KUKA KRL program: wkz1_ok.src, wkz1_ok.dat

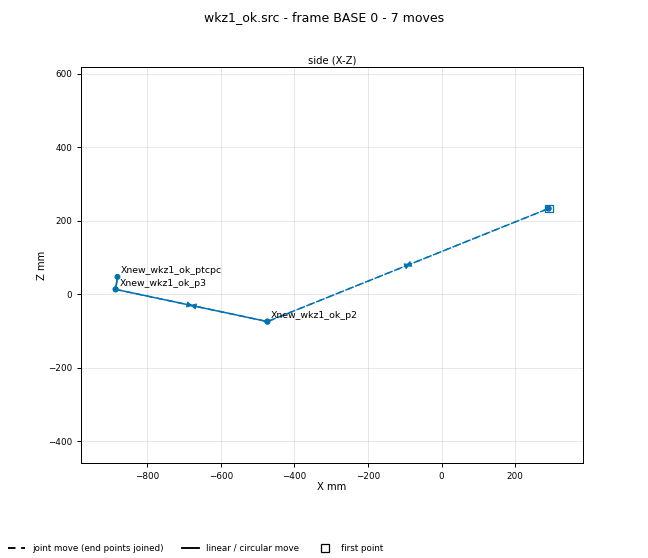
[picture p0: tool path of wkz1_ok.src in frame BASE 0, 7 of 9 moves have a stored position in this frame; points joined in program order, loops and branches not executed]
--- wkz1_ok.src ---
&ACCESS RVP
&COMMENT CHK_TCP_C1
&PARAM DISKPATH = Program/FUNCIONANDO
DEF WKZ1_OK ( )

;# Include block for krc/r1/mada/$config.dat or r1/$config.dat
;# TOOL_DATA[1]={X 73.860,Y 19.790,Z 1095.269,A -165.0000,B -25.0000,C 180.0000}
;# End of Include block for krc/r1/mada/$config.dat or r1/$config.dat
;FOLD INI
  ;FOLD BASISTECH INI
    GLOBAL INTERRUPT DECL 3 WHEN $STOPMESS==TRUE DO IR_STOPM ( )
    INTERRUPT ON 3
    BAS (#INITMOV,0 )
  ;ENDFOLD (BASISTECH INI)
  ;FOLD USER INI
    ;Make your modifications here
  ;ENDFOLD (USER INI)
;ENDFOLD (INI)
;FOLD PTP HOME  Vel= 100 % DEFAULT;%{PE}%V3.2.0,%MKUKATPBASIS,%CMOVE,%VPTP,%P 1:PTP, 2:HOME, 3:, 5:100, 7:DEFAULT
$BWDSTART = FALSE
$H_POS=XHOME
PDAT_ACT=PDEFAULT
BAS (#PTP_DAT )
FDAT_ACT=FHOME
BAS (#FRAMES )
BAS (#VEL_PTP,100 )
PTP  XHOME
;ENDFOLD
;#END_HEADER

;# ============ START PATH : wkz1_ok =============

; Caracterização dos meios de produção:
; Versão Atual:
; 04/05/2013 12:00 Name: P13.090-R6 CHANGES: Check TCP C1
chk_w1_wechs_ok ( )              ; CHECK GUN C1
;FOLD PTP new_wkz1_ok_p1  Vel=100 % P_OLP1 Tool[1]" " Base[0]  ;%{PE}%R8.3,%MKUKATPBASIS,%CMOVE,%VPTP,%P 1:PTP, 2:new_wkz1_ok_p1, 3:, 5:100, 7:P_OLP1
$BWDSTART = FALSE
PDAT_ACT= PP_OLP1
FDAT_ACT= Fnew_wkz1_ok_p1
BAS(#PTP_PARAMS,100)
PTP Xnew_wkz1_ok_p1
;ENDFOLD
;FOLD PTP new_wkz1_ok_p2  Vel=100 % P_OLP2 Tool[1]" " Base[0]  ;%{PE}%R8.3,%MKUKATPBASIS,%CMOVE,%VPTP,%P 1:PTP, 2:new_wkz1_ok_p2, 3:, 5:100, 7:P_OLP2
$BWDSTART = FALSE
PDAT_ACT= PP_OLP2
FDAT_ACT= Fnew_wkz1_ok_p2
BAS(#PTP_PARAMS,100)
PTP Xnew_wkz1_ok_p2
;ENDFOLD
;FOLD LIN new_wkz1_ok_p3  Vel=2.00 m/s L_OLP1 Tool[1]" " Base[0] ;%{PE}%R8.3,%MKUKATPBASIS,%CMOVE,%VLIN,%P 1:LIN, 2:new_wkz1_ok_p3, 3:, 5:2.00, 7:L_OLP1
$BWDSTART = FALSE
LDAT_ACT= LL_OLP1
FDAT_ACT= Fnew_wkz1_ok_p3
BAS(#CP_PARAMS,2.00)
LIN Xnew_wkz1_ok_p3
;ENDFOLD
;Ponto Check TCP
;FOLD LIN new_wkz1_ok_ptcpc  Vel=2.00 m/s L_OLP2 Tool[1]" " Base[0] ;%{PE}%R8.3,%MKUKATPBASIS,%CMOVE,%VLIN,%P 1:LIN, 2:new_wkz1_ok_ptcpc, 3:, 5:2.00, 7:L_OLP2
$BWDSTART = FALSE
LDAT_ACT= LL_OLP2
FDAT_ACT= Fnew_wkz1_ok_ptcpc
BAS(#CP_PARAMS,2.00)
LIN Xnew_wkz1_ok_ptcpc
;ENDFOLD
;FOLD WAIT Time= 3 sec;%{PE}%R8.3,%MKUKATPBASIS,%CWAIT,%VWAIT,%P 2:3
WAIT SEC 3
;ENDFOLD
;FOLD LIN new_wkz1_ok_p4  Vel=2.00 m/s L_OLP3 Tool[1]" " Base[0] ;%{PE}%R8.3,%MKUKATPBASIS,%CMOVE,%VLIN,%P 1:LIN, 2:new_wkz1_ok_p4, 3:, 5:2.00, 7:L_OLP3
$BWDSTART = FALSE
LDAT_ACT= LL_OLP3
FDAT_ACT= Fnew_wkz1_ok_p4
BAS(#CP_PARAMS,2.00)
LIN Xnew_wkz1_ok_p4
;ENDFOLD
;FOLD PTP new_wkz1_ok_p5  Vel=100 % P_OLP3 Tool[1]" " Base[0]  ;%{PE}%R8.3,%MKUKATPBASIS,%CMOVE,%VPTP,%P 1:PTP, 2:new_wkz1_ok_p5, 3:, 5:100, 7:P_OLP3
$BWDSTART = FALSE
PDAT_ACT= PP_OLP3
FDAT_ACT= Fnew_wkz1_ok_p5
BAS(#PTP_PARAMS,100)
PTP Xnew_wkz1_ok_p5
;ENDFOLD
;FOLD PTP new_wkz1_ok_p6  Vel=100 % P_OLP4 Tool[1]" " Base[0]  ;%{PE}%R8.3,%MKUKATPBASIS,%CMOVE,%VPTP,%P 1:PTP, 2:new_wkz1_ok_p6, 3:, 5:100, 7:P_OLP4
$BWDSTART = FALSE
PDAT_ACT= PP_OLP4
FDAT_ACT= Fnew_wkz1_ok_p6
BAS(#PTP_PARAMS,100)
PTP Xnew_wkz1_ok_p6
;ENDFOLD

;#START_TRAILER
;FOLD PTP HOME  Vel= 100 % DEFAULT;%{PE}%V3.2.0,%MKUKATPBASIS,%CMOVE,%VPTP,%P 1:PTP, 2:HOME, 3:, 5:100, 7:DEFAULT
$BWDSTART = FALSE
$H_POS=XHOME
PDAT_ACT=PDEFAULT
BAS (#PTP_DAT )
FDAT_ACT=FHOME
BAS (#FRAMES )
BAS (#VEL_PTP,100 )
PTP  XHOME
;ENDFOLD
END

--- wkz1_ok.dat ---
&ACCESS RVP
&COMMENT CHK_TCP_C1
&PARAM DISKPATH = Program/FUNCIONANDO
DEFDAT  wkz1_ok
;FOLD EXTERNAL DECLARATIONS;%{PE}%MKUKATPBASIS,%CEXT,%VCOMMON,%P
;FOLD BASISTECH EXT;%{PE}%MKUKATPBASIS,%CEXT,%VEXT,%P
EXT  BAS (BAS_COMMAND  :IN,REAL  :IN )
DECL INT SUCCESS
;ENDFOLD (BASISTECH EXT)
;FOLD USER EXT;%{E}%MKUKATPUSER,%CEXT,%VEXT,%P
;Make your modifications here
;ENDFOLD (USER EXT)
;ENDFOLD (EXTERNAL DECLARATIONS)

;# ============ START PATH : wkz1_ok =============
DECL FDAT Fnew_wkz1_ok_p1={TOOL_NO 1,BASE_NO 0,IPO_FRAME #BASE,POINT2[] " "}
DECL PDAT PP_OLP1={VEL 100.0,ACC 50.0,APO_DIST 0.0}
DECL E6POS Xnew_wkz1_ok_p1={X 291.243988,Y -1285.88794,Z 233.281006,A 13.0198002,B 2.4052,C 1.18589997,S 2,T 10}
DECL FDAT Fnew_wkz1_ok_p2={TOOL_NO 1,BASE_NO 0,IPO_FRAME #BASE,POINT2[] " "}
DECL PDAT PP_OLP2={VEL 100.0,ACC 50.0,APO_DIST 0.0}
DECL E6POS Xnew_wkz1_ok_p2={X -473.602997,Y -1280.02002,Z -74.2460022,A 146.021698,B -0.95389998,C -2.53250003,S 2,T 2}
DECL FDAT Fnew_wkz1_ok_p3={TOOL_NO 1,BASE_NO 0,IPO_FRAME #BASE,POINT2[] " "}
DECL E6POS Xnew_wkz1_ok_p3={X -886.51001,Y -1289.66003,Z 13.3669996,A 171.756897,B -2.65339994,C -0.53549999,S 2,T 2}
DECL LDAT LL_OLP1={VEL 2.0,ACC 100.0,APO_DIST 0.0,APO_FAC 0.0,ORI_TYP #VAR,CIRC_TYP #BASE,JERK_FAC 50.0}
DECL FDAT Fnew_wkz1_ok_ptcpc={TOOL_NO 1,BASE_NO 0,IPO_FRAME #BASE,POINT2[] " "}
DECL E6POS Xnew_wkz1_ok_ptcpc={X -881.550415,Y -1291.69397,Z 47.3409119,A 171.412704,B -2.65365791,C -0.829671085,S 18,T 2,E1 0.0,E2 0.0,E3 0.0,E4 0.0,E5 0.0,E6 0.0}
DECL LDAT LL_OLP2={VEL 2.0,ACC 100.0,APO_DIST 0.0,APO_FAC 0.0,ORI_TYP #VAR,CIRC_TYP #BASE,JERK_FAC 50.0}
DECL FDAT Fnew_wkz1_ok_p4={TOOL_NO 1,BASE_NO 0,IPO_FRAME #BASE,POINT2[] " "}
DECL E6POS Xnew_wkz1_ok_p4={X -886.51001,Y -1289.66003,Z 13.3669996,A 171.756897,B -2.65339994,C -0.53549999,S 2,T 2}
DECL LDAT LL_OLP3={VEL 2.0,ACC 100.0,APO_DIST 0.0,APO_FAC 0.0,ORI_TYP #VAR,CIRC_TYP #BASE,JERK_FAC 50.0}
DECL FDAT Fnew_wkz1_ok_p5={TOOL_NO 1,BASE_NO 0,IPO_FRAME #BASE,POINT2[] " "}
DECL PDAT PP_OLP3={VEL 100.0,ACC 50.0,APO_DIST 0.0}
DECL E6POS Xnew_wkz1_ok_p5={X -473.602997,Y -1280.02002,Z -74.2460022,A 146.021698,B -0.95389998,C -2.53250003,S 2,T 2}
DECL FDAT Fnew_wkz1_ok_p6={TOOL_NO 1,BASE_NO 0,IPO_FRAME #BASE,POINT2[] " "}
DECL PDAT PP_OLP4={VEL 100.0,ACC 50.0,APO_DIST 0.0}
DECL E6POS Xnew_wkz1_ok_p6={X 291.243988,Y -1285.88794,Z 233.281006,A 13.0198002,B 2.4052,C 1.18589997,S 2,T 10}
ENDDAT
